// TIA Portal V16 export
// export: Created 2021-11-12T13:33:01.0256083Z, ExportSetting WithDefaults, DisplayName Totally Integrated Automation Portal, DisplayVersion V16 Update 3, DisplayName TIA Portal Version Control Interface, DisplayVersion V16 Update 2, DisplayName TIA Portal Openness, DisplayVersion V16 Update 3, DisplayName SINAMICS Startdrive Advanced, DisplayVersion V16 Update 5, DisplayName SINAMICS Startdrive G130, G150, S120, S150, SINAMICS MV, S210, DisplayVersion V16 Update 5, DisplayName SINAMICS Startdrive G110M, G120, G120C, G120D, G120P, G115D, DisplayVersion V16 Update 5, DisplayName STEP 7 Professional, DisplayVersion V16 Update 3, DisplayName STEP 7 Safety, DisplayVersion V16, DisplayName WinCC UA Professional, DisplayVersion V16 Update 3
DATA_BLOCK "HMI_PARAM_420"   // DB103
{ S7_Optimized_Access := 'TRUE' }
VERSION : 0.1
// stored: AutoNumber true, DBAccessibleFromOPCUA true, IsOnlyStoredInLoadMemory false, IsRetainMemResEnabled false, IsWriteProtectedInAS false, MemoryReserve 100
   VAR
      xxxxx___BinarySensors___xxxxx_1 : Byte;
      "EQ01-BL01" : "UDT_CH_DI_Parameter";   // Sensor for min surface (LSL1442) / Hladina min (LSL1442)
      "EQ01-BL02" : "UDT_CH_DI_Parameter";   // Sensor for max surface (LSH1443) / Hladina max (LSH1443)
      "EQ01-MA02_20" : "UDT_CH_DI_Parameter";   // Valve (A1418) - closed
      "EQ01-MA02_24" : "UDT_CH_DI_Parameter";   // Valve (A1418) - opened
      "EQ01-MA03_20" : "UDT_CH_DI_Parameter";   // Valve (A1415) - closed
      "EQ01-MA03_24" : "UDT_CH_DI_Parameter";   // Valve (A1415) - opened
      "EQ01-MA04_20" : "UDT_CH_DI_Parameter";   // Valve (A1412) - closed
      "EQ01-MA04_24" : "UDT_CH_DI_Parameter";   // Valve (A1412) - opened
      xxxxx___BinaryOthers___xxxxx_1 : Byte;
      "UC10-FC21_14" : "UDT_CH_DI_Parameter";   // 230V Hardening tube / 230V Zachlazovací nádrž
      "UC11-FC01_14" : "UDT_CH_DI_Parameter";   // 400V Pump of circulation P32 OK / 400V Čerpadlo cirkulace P32 OK
      xxxxx___AnalogueSensors___xxxxx_1 : Byte;
   END_VAR
   VAR RETAIN
      "EQ01-BT01" : "UDT_CH_AI_Parameter";   // Temperature measurment (TIC 1424) / Měření teploty (TIC 1425)
      "EQ01-BP01" : "UDT_CH_AI_Parameter";   // Tenzometric sond for measure surface (LIC 1430) / Tenzometrická sonda pro měření hladiny(LIC 1431)
      "EQ01-MA03_81" : "UDT_CH_AI_Parameter";   // Meření ventilu A 1415 Zavřeno - otevřeno
   END_VAR
   VAR
      xxxxx___Drives___xxxxx_1 : Byte;
      "EQ01-MA01" : "UDT_Drive1_Parameter";   // Pump of circulation (P32) / Čerpadlo cirkulace (P32)
      "EQ01-MA02" : "UDT_Valve2WB_Parameter";   // Valve with servomotor (A1418) / Ventil se servopohonem (A1418)
      "EQ01-MA03" : "UDT_Valve2WB_Parameter";   // Valve with servomotor (A1415) / Ventil se servopohonem (A1415)
      "EQ01-MA04" : "UDT_Valve2WB_Parameter";   // Valve with servomotor (A1412) / Ventil se servopohonem (A1412)
   END_VAR
   VAR RETAIN
      "UC11-TA01" : "UDT_SINAMICS_G120_Parameter";   // Frequence changer ( pro P32) / Frekvenční měnič ( pro P32)
   END_VAR
   VAR
      xxxxx___Alarms___xxxxx : Byte;
      ES : "UDT_DI_Mon_Parameter";   // E-stop
      KF31 : "UDT_DI_Mon_Parameter";   // module KF31
      Alarm_1 { S7_SetPoint := 'True'} : "UDT_DI_Mon_Parameter";   // Sensor Max level active and sensor Min level
      Alarm_2 { S7_SetPoint := 'True'} : "UDT_DI_Mon_Parameter";   // Sensor Min level active and analog level sensor under 10%
      Alarm_3 { S7_SetPoint := 'True'} : "UDT_DI_Mon_Parameter";   // Analog level sensor over 40% and sensor min level not active
      Alarm_4 { S7_SetPoint := 'True'} : "UDT_DI_Mon_Parameter";   // Water temperature high
      Alarm_5 { S7_SetPoint := 'True'} : "UDT_DI_Mon_Parameter";   // Water temperature low
      Alarm_6 { S7_SetPoint := 'True'} : "UDT_DI_Mon_Parameter";   // Water level high
      Alarm_7 { S7_SetPoint := 'True'} : "UDT_DI_Mon_Parameter";   // BSN3 tacts and water level NOK
      Alarm_8 { S7_SetPoint := 'True'} : "UDT_DI_Mon_Parameter";   // Filling and no water level change
      Alarm_9 { S7_SetPoint := 'True'} : "UDT_DI_Mon_Parameter";   // Drain and no water level change
      xxxxx___Others___xxxxx { S7_SetPoint := 'True'} : Byte;
      "EQ01-MA03_RegPar" : Struct   // Cooling regulation
         PGain : Real := 1.0;
         Bias : Real := 50.0;
      END_STRUCT;
   END_VAR
BEGIN
   "EQ01-BT01".RawOvFlwLim := 29376;
   "EQ01-BT01".RawUnFlwLim := -1728;
   "EQ01-BT01".RMax := 100.0;
   "EQ01-BT01".RMin := 0.0;
   "EQ01-BP01".RawMax := 4540;
   "EQ01-BP01".RawOvFlwLim := 29376;
   "EQ01-BP01".RawUnFlwLim := -1728;
   "EQ01-BP01".RMax := 100.0;
   "EQ01-BP01".RMin := 0.0;
   "EQ01-MA03_81".RMax := 100.0;
   "EQ01-MA03_81".RMin := 0.0;
   "UC11-TA01".RefSpdP2000 := 3000.0;
   "UC11-TA01".RefCurrP2002 := 16.5;
   "UC11-TA01".RefTrqP2003 := 35.85;
END_DATA_BLOCK
